(* Logix 5000 project; controller PRU vendor 1 type 14 code 107 rev 20.13; software revision 20.01; part 16 of 17 *)
(* tags used below, declared in another part *)
   ABS_ENCODER_ERROR_MINUS : REAL;
   ABS_ENCODER_ERROR_PLUS : REAL;
   ACCEL_DECEL_RAMP : REAL;   // VFD Accel/Decel ramp rate * 10ms ie 100 * 10ms = 1sec
   ACTUAL_FWD_ION : BOOL;
   ACTUAL_ILLEGAL_ION : BOOL;
   ACTUAL_REV_ION : BOOL;
   AFI : BOOL;
   AUTO_FWD_CMD : BOOL;
   AUTO_FWD_CMD_GON : BOOL;
   AUTO_FWD_CMD_GON_VALUE : DINT;
   AUTO_FWD_CMD_VALUE : DINT;
   CENTERING_BON : BOOL;
   CENTERING_BON_ONS : BOOL;
   CENTERING_BON_SS : BOOL;
   CENTERING_ERROR : REAL;
   CENTERING_ERROR_NOW : REAL;
   CENTERING_ERROR_WAS : REAL;
   CENTERING_ONS : BOOL;
   CENTERING_SS : BOOL;
   CENTERING_TON : TIMER;
   CR7_VFD_DRYERL_GON : BOOL;
   CR7_VFD_DRYERL_LON : BOOL;
   DATA_RECORD_INDEX : INT;
   DRYER : DUAL_SCREW;
   DRYER_CENTER_STARTUP_MODE : BOOL;
   DRYER_IS_CENTERING : BOOL;
   DRYER_MODE_AUTO : BOOL;
   DRYERL_ACTUAL_SPEED : REAL;
   DRYERR_ACTUAL_SPEED : REAL;
   ENCODER_ACC : REAL;
   ENCODER_ERROR : REAL;
   ENCODER_OFFSET : REAL;
   ENCODER_RATE : REAL;
   ESR_CONTACT_1_ION : BOOL;
   ESR_CONTACT_2_ION : BOOL;
   ESR_RESET_PB_ION : BOOL;
   FAULT : DINT[100];
   FAULT_31_14_ONS : BOOL;
   FAULT_TIMER : TIMER[10000];
   FAULT_TIMER_3112_TmrExtended : BOOL;
   FAULT_TIMER_3112_TmrNormal : BOOL;
   FAULTS_FA1_IOK : BOOL;   // SYSTEM LEVEL FAULTS ARE OK.
   FAULTS_FA1B_IOK : BOOL;   // STOP PUSHBUTTON FAULTS ARE OK.
   FAULTS_FA3_IOK : BOOL;
   FAULTS_FA3A_IOK : BOOL;   // SCREWS DRIVES NOT FAULTED.
   FAULTS_FA3B_IOK : BOOL;   // ENCODERS NOT FAULTED.
   FEED_TIME_OFF : TIMER;
   FEED_TIME_OFF_REM : REAL;
   FEED_TIME_OFF_REM_TEMP : REAL;
   FEED_TIME_OFF_SEC : REAL;
   FEED_TIME_ON : TIMER;
   FEED_TIME_ON_REM : REAL;
   FEED_TIME_ON_REM_TEMP : REAL;
   FEED_TIME_ON_SEC : REAL;
   FEED_TRIGGER : BOOL;
   FWD_CMD_BON : TIMER;
   GRAY : REAL[4097];
   HMI_ALARM_RESET : BOOL;
   HMI_AUTO_SETPOINT_FDBK : REAL;
   HMI_CR7_FORCE_OFF : BOOL;
   HMI_CR7_FORCE_ON : BOOL;
   HMI_DCS_SPEED_FDBK : REAL;
   HMI_DSC_SPEED_CMD : REAL;
   HMI_FINAL_SCREW_POSITION_ERROR : REAL;
   HMI_OSC_INC : REAL;
   HMI_WIPER_OSC_SETPOINT : REAL;
   HMI_ZERO_SPEED_FORCE_ION : BOOL;
   INTERRUPT_INDEX : INT;
   LEFT_AUTO_PCNT_SETPOINT : REAL;
   LEFT_RATE : REAL;
   MASTER_RIGHT_CMD : BOOL;
   MAX_ENCODER_ERROR_MINUS : REAL;
   MAX_ENCODER_ERROR_PLUS : REAL;
   MIX_FWD_PRESET : REAL;
   MIX_MODE_TIMEBASE : BOOL;
   MIX_REV_PER_MIN : REAL;
   MIX_REV_PRESET : REAL;
   MODE_DRYER : INT;
   OK_TO_CHANGE_DIR : BOOL;
   OK_TO_STOP : BOOL;
   PF70EL_Message : MESSAGE;
   PF70ER_Message : MESSAGE;
   RAMP_COUNT : DINT;
   RAMP_TIME : DINT;
   RAMPING_SPEED_DOWN : BOOL;
   RAMPING_SPEED_UP : BOOL;
   RelaxEncoderFaultTime_SpeedSP : REAL;
   RelaxEncoderFaultTime_SpeedSP_Rev : REAL;
   RETENTION_TIME_MIN : REAL;
   REV_CMD_BON : TIMER;
   RIGHT_AUTO_PCNT_SETPOINT : REAL;
   RIGHT_RATE : REAL;
   SCREW_ENCODERS : SCREW_ENCODERS;
   SCREW_PITCH_CONSTANT : REAL;
   SCREW_SPEED : SCREW_SPEED;
   SCREW_SPEED_OUT_L : REAL;
   SCREW_SPEED_OUT_R : REAL;
   SCREW_WIPE : SCREW_WIPER;
   SCREWS_ENABLE_GON : BOOL;   // Dryer screw faults are ok.
   SCREWS_WIPE_HOLD_TIME : DINT;
   SET_PYRO_SPEED_TO_ZERO : BOOL;
   SLAVE_COMP_LIMIT : REAL;
   SPEED_RAMP_FREEZE_TOF : TIMER;
   SPEED_RAMP_MULT : REAL;
   VFD_1_Current : DINT;
   VFD_1_Current_Real : REAL;
   VFD_1_Tot : EnergyTot;   // Left Dryer
   VFD_2_Current : DINT;
   VFD_2_Current_Real : REAL;
   VFD_2_Tot : EnergyTot;   // Right Dryer
   VFDS_BON : BOOL;   // DRYER VFDs HAVE BEEN COMMANDED ON FOR 1 SECOND.
   WIPE_ACTUAL : REAL;
   WIPE_EON : BOOL;
   WIPE_FREEZE_CMD : BOOL;
   WIPE_HOLDING : BOOL;
   WIPE_MASTER : BOOL;
   WIPE_MASTER_BOF : TIMER;
   WIPE_MASTER_BON : TIMER;
   WIPE_MASTER_ONS : BOOL;
   WIPE_MASTER_SS : BOOL;
   WIPE_PERIOD_COUNTS_ACC : REAL;
   WIPE_PERIOD_ONS : BOOL;
   WIPE_PERIOD_SECONDS : REAL;
   WIPE_TON : TIMER;
(* SCREW_CONTROL, continued *)

ROUTINE B03_FA3_B_ENCODER_FAULTS_3100   (* ladder *)
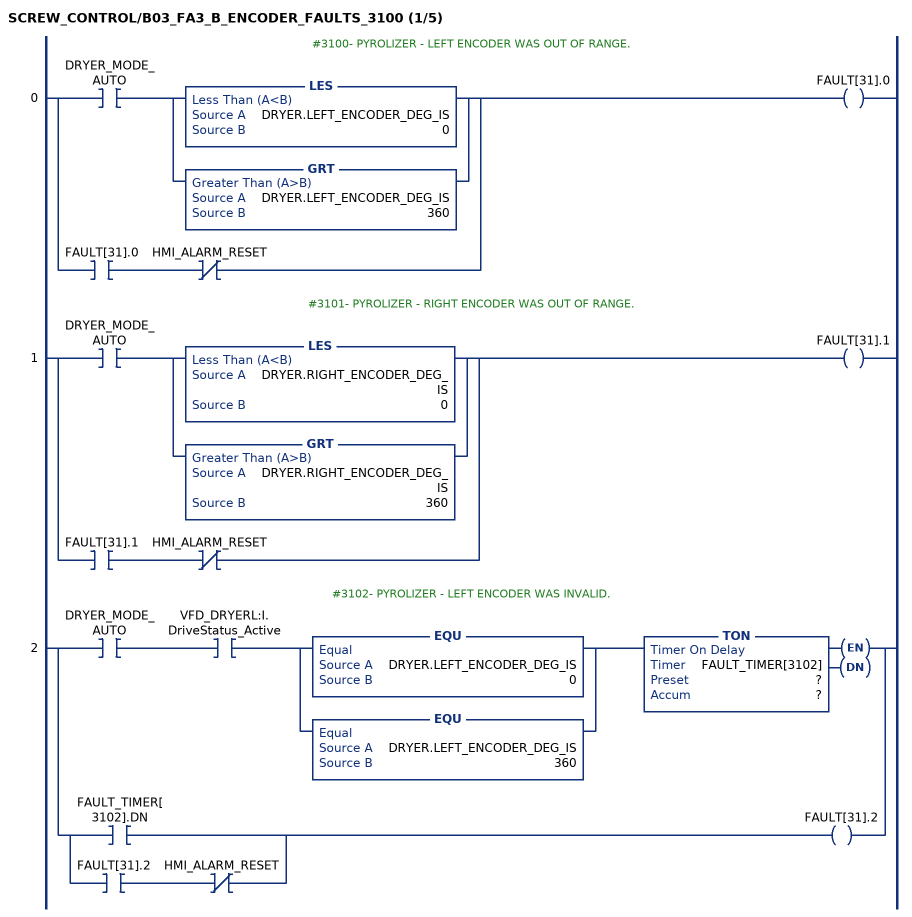
   // #3100- PYROLIZER - LEFT ENCODER WAS OUT OF RANGE.
   0: [XIC(DRYER_MODE_AUTO) [LES(DRYER.LEFT_ENCODER_DEG_IS,0) ,GRT(DRYER.LEFT_ENCODER_DEG_IS,360) ] ,XIC(FAULT[31].0) XIO(HMI_ALARM_RESET) ]OTE(FAULT[31].0);
   // #3101- PYROLIZER - RIGHT ENCODER WAS OUT OF RANGE.
   1: [XIC(DRYER_MODE_AUTO) [LES(DRYER.RIGHT_ENCODER_DEG_IS,0) ,GRT(DRYER.RIGHT_ENCODER_DEG_IS,360) ] ,XIC(FAULT[31].1) XIO(HMI_ALARM_RESET) ]OTE(FAULT[31].1);
   // #3102- PYROLIZER - LEFT ENCODER WAS INVALID.
   2: [XIC(DRYER_MODE_AUTO) XIC(VFD_DRYERL:I.DriveStatus_Active) [EQU(DRYER.LEFT_ENCODER_DEG_IS,0) ,EQU(DRYER.LEFT_ENCODER_DEG_IS,360) ] TON(FAULT_TIMER[3102],?,?) ,[XIC(FAULT_TIMER[3102].DN) ,XIC(FAULT[31].2) XIO(HMI_ALARM_RESET) ] OTE(FAULT[31].2) ];
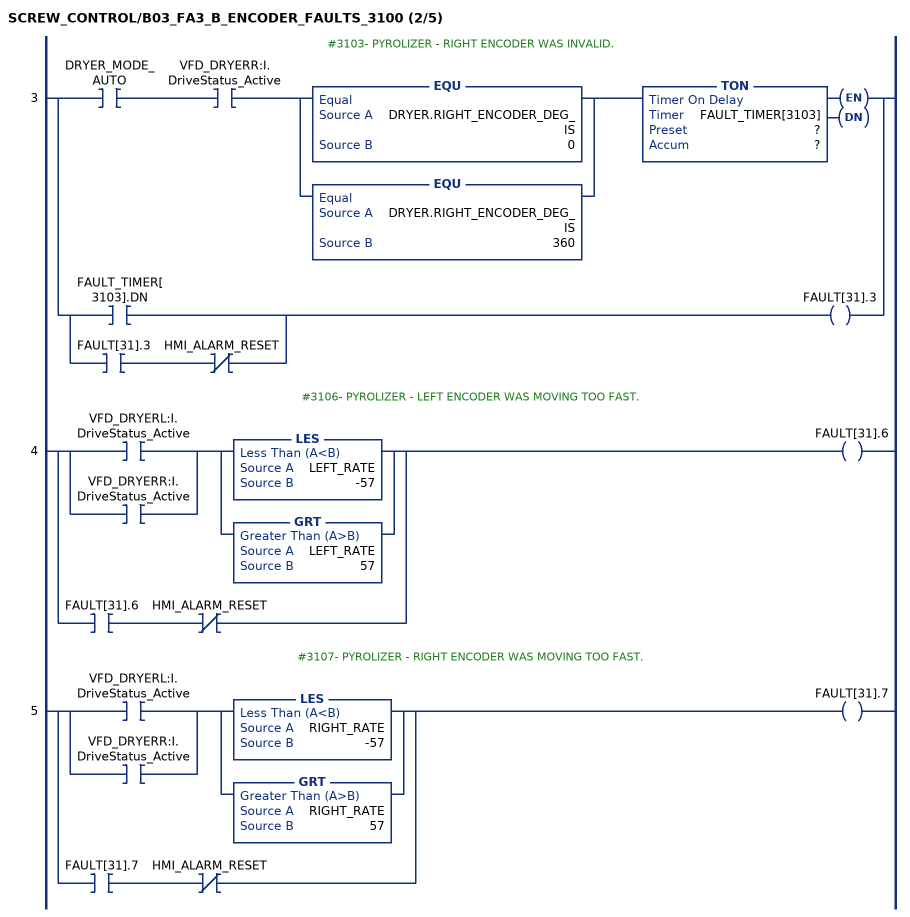
   // #3103- PYROLIZER - RIGHT ENCODER WAS INVALID.
   3: [XIC(DRYER_MODE_AUTO) XIC(VFD_DRYERR:I.DriveStatus_Active) [EQU(DRYER.RIGHT_ENCODER_DEG_IS,0) ,EQU(DRYER.RIGHT_ENCODER_DEG_IS,360) ] TON(FAULT_TIMER[3103],?,?) ,[XIC(FAULT_TIMER[3103].DN) ,XIC(FAULT[31].3) XIO(HMI_ALARM_RESET) ] OTE(FAULT[31].3) ];
   // #3106- PYROLIZER - LEFT ENCODER WAS MOVING TOO FAST.
   4: [[XIC(VFD_DRYERL:I.DriveStatus_Active) ,XIC(VFD_DRYERR:I.DriveStatus_Active) ] [LES(LEFT_RATE,-57) ,GRT(LEFT_RATE,57) ] ,XIC(FAULT[31].6) XIO(HMI_ALARM_RESET) ]OTE(FAULT[31].6);
   // #3107- PYROLIZER - RIGHT ENCODER WAS MOVING TOO FAST.
   5: [[XIC(VFD_DRYERL:I.DriveStatus_Active) ,XIC(VFD_DRYERR:I.DriveStatus_Active) ] [LES(RIGHT_RATE,-57) ,GRT(RIGHT_RATE,57) ] ,XIC(FAULT[31].7) XIO(HMI_ALARM_RESET) ]OTE(FAULT[31].7);
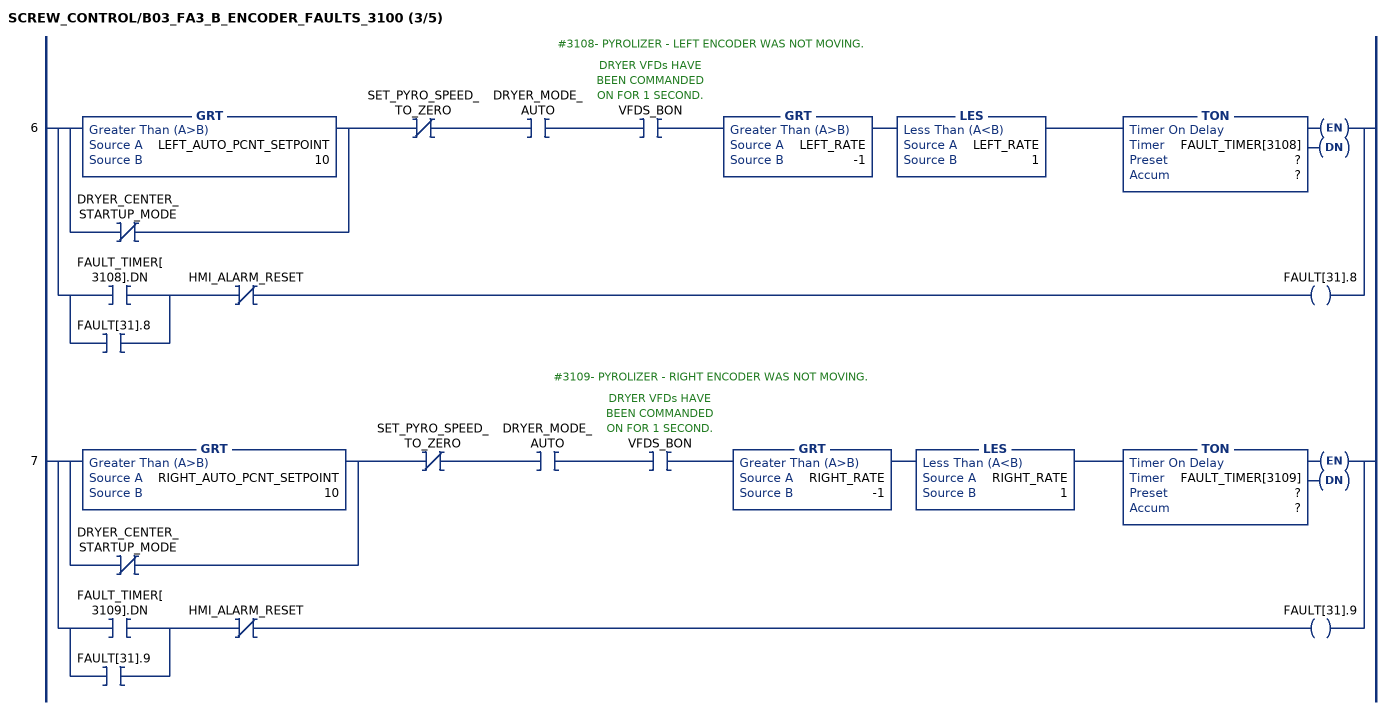
   // #3108- PYROLIZER - LEFT ENCODER WAS NOT MOVING.
   6: [[GRT(LEFT_AUTO_PCNT_SETPOINT,10) ,XIO(DRYER_CENTER_STARTUP_MODE) ] XIO(SET_PYRO_SPEED_TO_ZERO) XIC(DRYER_MODE_AUTO) XIC(VFDS_BON) GRT(LEFT_RATE,-1) LES(LEFT_RATE,1) TON(FAULT_TIMER[3108],?,?) ,[XIC(FAULT_TIMER[3108].DN) ,XIC(FAULT[31].8) ] XIO(HMI_ALARM_RESET) OTE(FAULT[31].8) ];
   // #3109- PYROLIZER - RIGHT ENCODER WAS NOT MOVING.
   7: [[GRT(RIGHT_AUTO_PCNT_SETPOINT,10) ,XIO(DRYER_CENTER_STARTUP_MODE) ] XIO(SET_PYRO_SPEED_TO_ZERO) XIC(DRYER_MODE_AUTO) XIC(VFDS_BON) GRT(RIGHT_RATE,-1) LES(RIGHT_RATE,1) TON(FAULT_TIMER[3109],?,?) ,[XIC(FAULT_TIMER[3109].DN) ,XIC(FAULT[31].9) ] XIO(HMI_ALARM_RESET) OTE(FAULT[31].9) ];
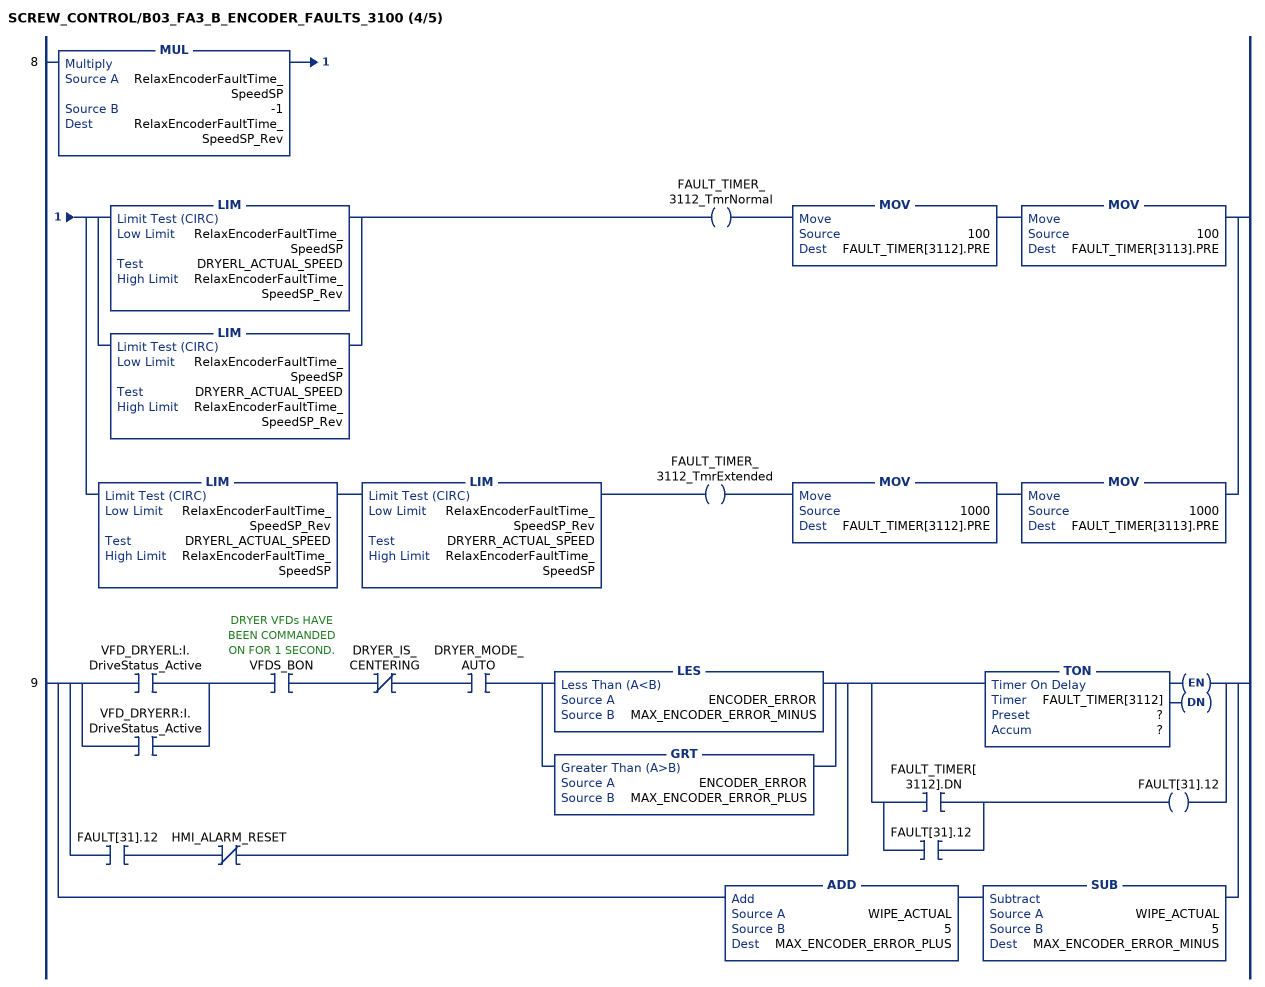
   8: MUL(RelaxEncoderFaultTime_SpeedSP,-1,RelaxEncoderFaultTime_SpeedSP_Rev)[[LIM(RelaxEncoderFaultTime_SpeedSP,DRYERL_ACTUAL_SPEED,RelaxEncoderFaultTime_SpeedSP_Rev) ,LIM(RelaxEncoderFaultTime_SpeedSP,DRYERR_ACTUAL_SPEED,RelaxEncoderFaultTime_SpeedSP_Rev) ] OTE(FAULT_TIMER_3112_TmrNormal) MOV(100,FAULT_TIMER[3112].PRE) MOV(100,FAULT_TIMER[3113].PRE) ,LIM(RelaxEncoderFaultTime_SpeedSP_Rev,DRYERL_ACTUAL_SPEED,RelaxEncoderFaultTime_SpeedSP) LIM(RelaxEncoderFaultTime_SpeedSP_Rev,DRYERR_ACTUAL_SPEED,RelaxEncoderFaultTime_SpeedSP) OTE(FAULT_TIMER_3112_TmrExtended) MOV(1000,FAULT_TIMER[3112].PRE) MOV(1000,FAULT_TIMER[3113].PRE) ];
   9: [[[XIC(VFD_DRYERL:I.DriveStatus_Active) ,XIC(VFD_DRYERR:I.DriveStatus_Active) ] XIC(VFDS_BON) XIO(DRYER_IS_CENTERING) XIC(DRYER_MODE_AUTO) [LES(ENCODER_ERROR,MAX_ENCODER_ERROR_MINUS) ,GRT(ENCODER_ERROR,MAX_ENCODER_ERROR_PLUS) ] ,XIC(FAULT[31].12) XIO(HMI_ALARM_RESET) ] [TON(FAULT_TIMER[3112],?,?) ,[XIC(FAULT_TIMER[3112].DN) ,XIC(FAULT[31].12) ] OTE(FAULT[31].12) ] ,ADD(WIPE_ACTUAL,5,MAX_ENCODER_ERROR_PLUS) SUB(WIPE_ACTUAL,5,MAX_ENCODER_ERROR_MINUS) ];
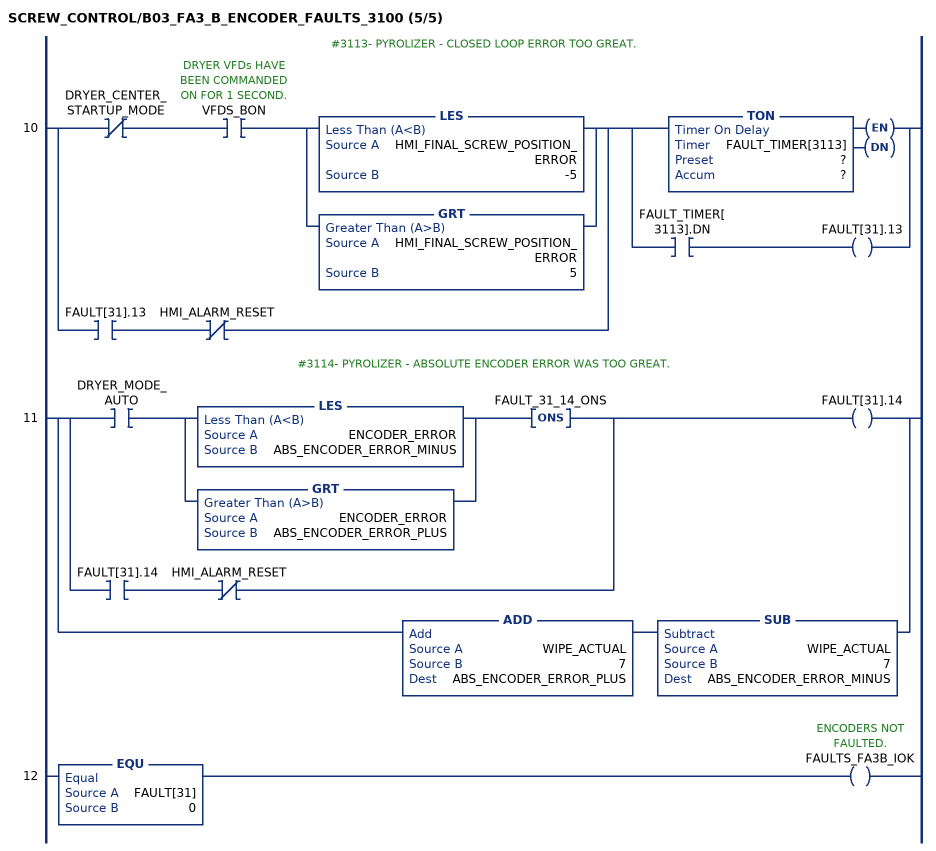
   // #3113- PYROLIZER - CLOSED LOOP ERROR TOO GREAT.
   10: [XIO(DRYER_CENTER_STARTUP_MODE) XIC(VFDS_BON) [LES(HMI_FINAL_SCREW_POSITION_ERROR,-5) ,GRT(HMI_FINAL_SCREW_POSITION_ERROR,5) ] ,XIC(FAULT[31].13) XIO(HMI_ALARM_RESET) ][TON(FAULT_TIMER[3113],?,?) ,XIC(FAULT_TIMER[3113].DN) OTE(FAULT[31].13) ];
   // #3114- PYROLIZER - ABSOLUTE ENCODER ERROR WAS TOO GREAT.
   11: [[XIC(DRYER_MODE_AUTO) [LES(ENCODER_ERROR,ABS_ENCODER_ERROR_MINUS) ,GRT(ENCODER_ERROR,ABS_ENCODER_ERROR_PLUS) ] ONS(FAULT_31_14_ONS) ,XIC(FAULT[31].14) XIO(HMI_ALARM_RESET) ] OTE(FAULT[31].14) ,ADD(WIPE_ACTUAL,7,ABS_ENCODER_ERROR_PLUS) SUB(WIPE_ACTUAL,7,ABS_ENCODER_ERROR_MINUS) ];
   12: EQU(FAULT[31],0)OTE(FAULTS_FA3B_IOK);
END_ROUTINE

ROUTINE DUALSCREW   (* ladder *)
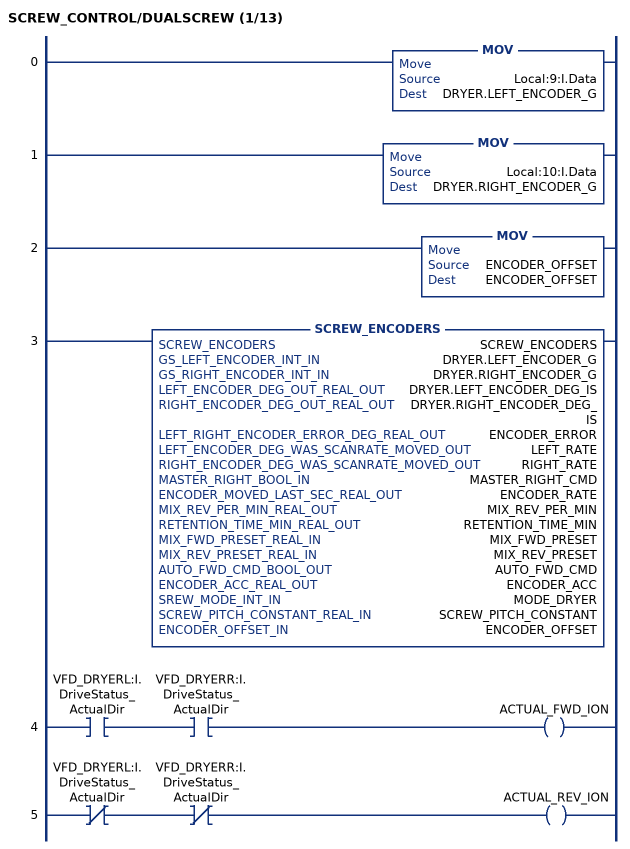
   0: MOV(Local:9:I.Data,DRYER.LEFT_ENCODER_G);
   1: MOV(Local:10:I.Data,DRYER.RIGHT_ENCODER_G);
   2: MOV(ENCODER_OFFSET,ENCODER_OFFSET);
   3: SCREW_ENCODERS(SCREW_ENCODERS,DRYER.LEFT_ENCODER_G,DRYER.RIGHT_ENCODER_G,DRYER.LEFT_ENCODER_DEG_IS,DRYER.RIGHT_ENCODER_DEG_IS,ENCODER_ERROR,LEFT_RATE,RIGHT_RATE,MASTER_RIGHT_CMD,ENCODER_RATE,MIX_REV_PER_MIN,RETENTION_TIME_MIN,MIX_FWD_PRESET,MIX_REV_PRESET,AUTO_FWD_CMD,ENCODER_ACC,MODE_DRYER,SCREW_PITCH_CONSTANT,ENCODER_OFFSET);
   4: XIC(VFD_DRYERL:I.DriveStatus_ActualDir)XIC(VFD_DRYERR:I.DriveStatus_ActualDir)OTE(ACTUAL_FWD_ION);
   5: XIO(VFD_DRYERL:I.DriveStatus_ActualDir)XIO(VFD_DRYERR:I.DriveStatus_ActualDir)OTE(ACTUAL_REV_ION);
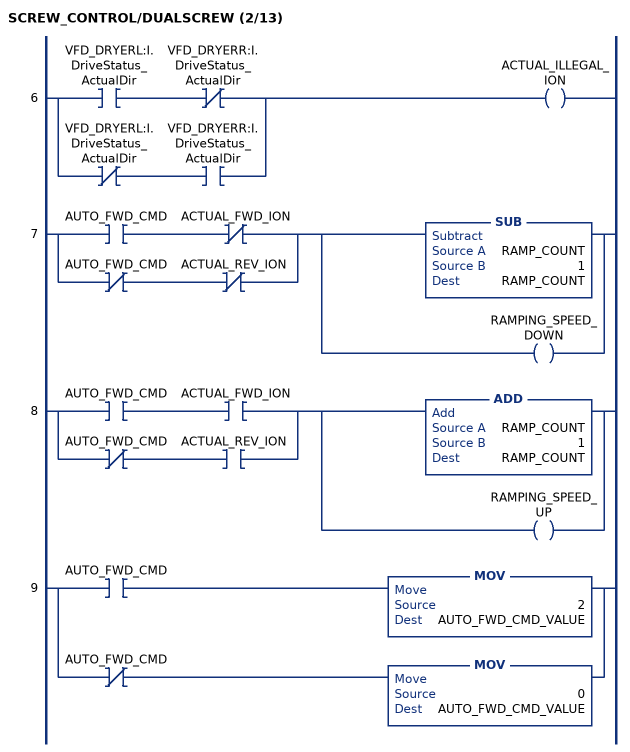
   6: [XIC(VFD_DRYERL:I.DriveStatus_ActualDir) XIO(VFD_DRYERR:I.DriveStatus_ActualDir) ,XIO(VFD_DRYERL:I.DriveStatus_ActualDir) XIC(VFD_DRYERR:I.DriveStatus_ActualDir) ]OTE(ACTUAL_ILLEGAL_ION);
   7: [XIC(AUTO_FWD_CMD) XIO(ACTUAL_FWD_ION) ,XIO(AUTO_FWD_CMD) XIO(ACTUAL_REV_ION) ][SUB(RAMP_COUNT,1,RAMP_COUNT) ,OTE(RAMPING_SPEED_DOWN) ];
   8: [XIC(AUTO_FWD_CMD) XIC(ACTUAL_FWD_ION) ,XIO(AUTO_FWD_CMD) XIC(ACTUAL_REV_ION) ][ADD(RAMP_COUNT,1,RAMP_COUNT) ,OTE(RAMPING_SPEED_UP) ];
   9: [XIC(AUTO_FWD_CMD) MOV(2,AUTO_FWD_CMD_VALUE) ,XIO(AUTO_FWD_CMD) MOV(0,AUTO_FWD_CMD_VALUE) ];
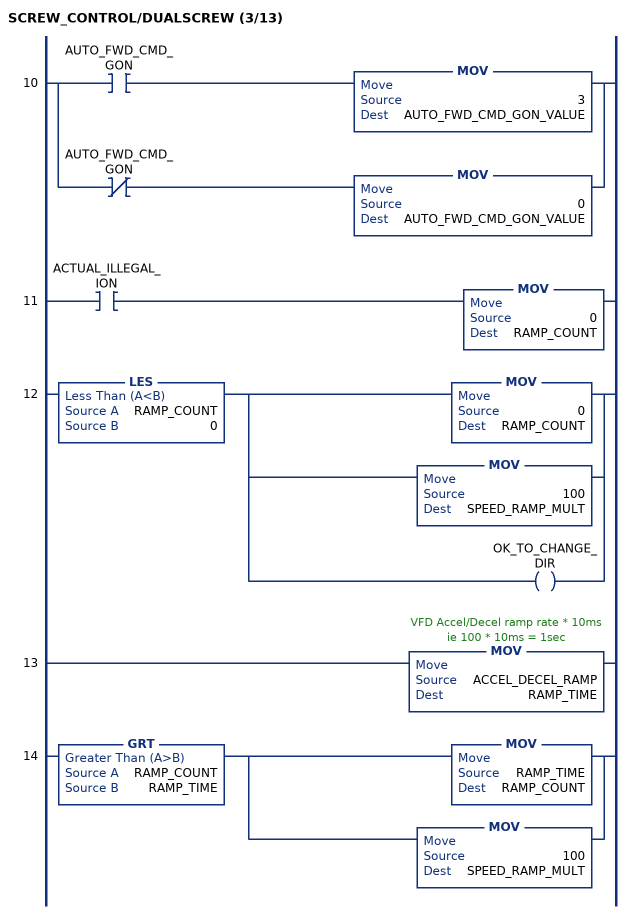
   10: [XIC(AUTO_FWD_CMD_GON) MOV(3,AUTO_FWD_CMD_GON_VALUE) ,XIO(AUTO_FWD_CMD_GON) MOV(0,AUTO_FWD_CMD_GON_VALUE) ];
   11: XIC(ACTUAL_ILLEGAL_ION)MOV(0,RAMP_COUNT);
   12: LES(RAMP_COUNT,0)[MOV(0,RAMP_COUNT) ,MOV(100,SPEED_RAMP_MULT) ,OTE(OK_TO_CHANGE_DIR) ];
   13: MOV(ACCEL_DECEL_RAMP,RAMP_TIME);
   14: GRT(RAMP_COUNT,RAMP_TIME)[MOV(RAMP_TIME,RAMP_COUNT) ,MOV(100,SPEED_RAMP_MULT) ];
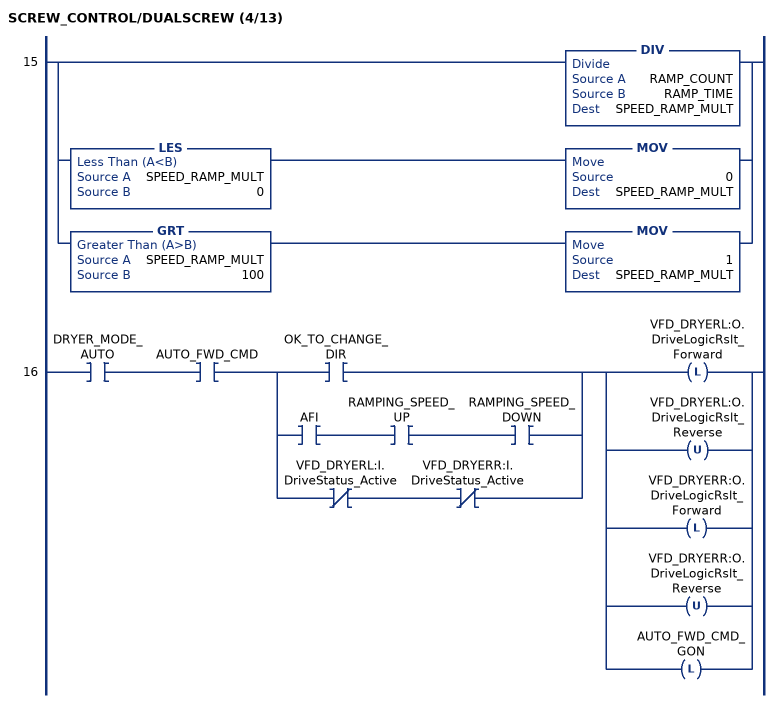
   15: [DIV(RAMP_COUNT,RAMP_TIME,SPEED_RAMP_MULT) ,LES(SPEED_RAMP_MULT,0) MOV(0,SPEED_RAMP_MULT) ,GRT(SPEED_RAMP_MULT,100) MOV(1,SPEED_RAMP_MULT) ];
   16: XIC(DRYER_MODE_AUTO)XIC(AUTO_FWD_CMD)[XIC(OK_TO_CHANGE_DIR) ,XIC(AFI) XIC(RAMPING_SPEED_UP) XIC(RAMPING_SPEED_DOWN) ,XIO(VFD_DRYERL:I.DriveStatus_Active) XIO(VFD_DRYERR:I.DriveStatus_Active) ][OTL(VFD_DRYERL:O.DriveLogicRslt_Forward) ,OTU(VFD_DRYERL:O.DriveLogicRslt_Reverse) ,OTL(VFD_DRYERR:O.DriveLogicRslt_Forward) ,OTU(VFD_DRYERR:O.DriveLogicRslt_Reverse) ,OTL(AUTO_FWD_CMD_GON) ];
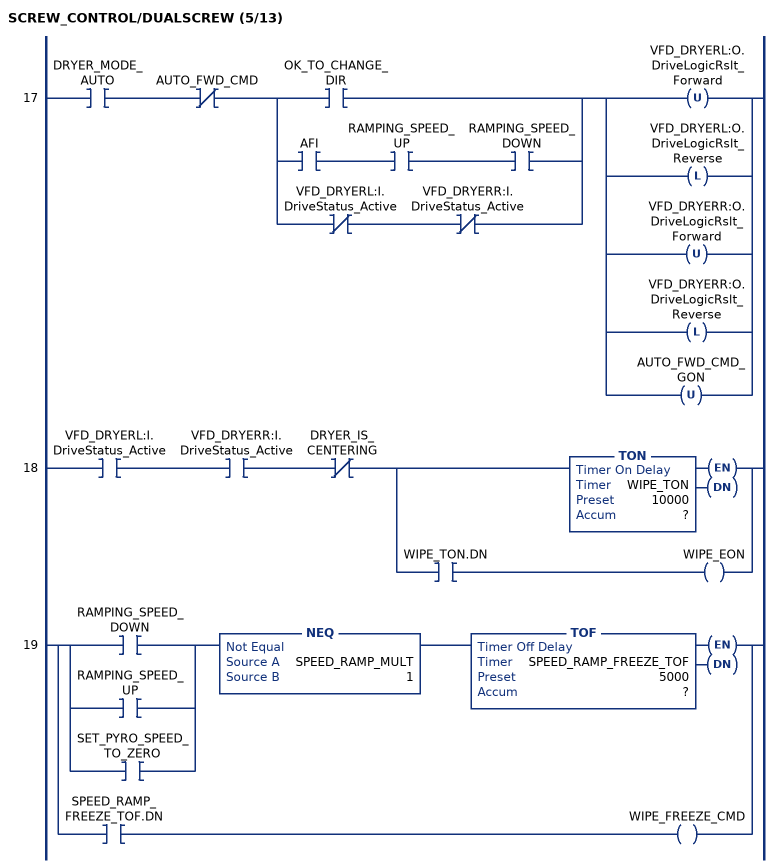
   17: XIC(DRYER_MODE_AUTO)XIO(AUTO_FWD_CMD)[XIC(OK_TO_CHANGE_DIR) ,XIC(AFI) XIC(RAMPING_SPEED_UP) XIC(RAMPING_SPEED_DOWN) ,XIO(VFD_DRYERL:I.DriveStatus_Active) XIO(VFD_DRYERR:I.DriveStatus_Active) ][OTU(VFD_DRYERL:O.DriveLogicRslt_Forward) ,OTL(VFD_DRYERL:O.DriveLogicRslt_Reverse) ,OTU(VFD_DRYERR:O.DriveLogicRslt_Forward) ,OTL(VFD_DRYERR:O.DriveLogicRslt_Reverse) ,OTU(AUTO_FWD_CMD_GON) ];
   18: XIC(VFD_DRYERL:I.DriveStatus_Active)XIC(VFD_DRYERR:I.DriveStatus_Active)XIO(DRYER_IS_CENTERING)[TON(WIPE_TON,?,?) ,XIC(WIPE_TON.DN) OTE(WIPE_EON) ];
   19: [[XIC(RAMPING_SPEED_DOWN) ,XIC(RAMPING_SPEED_UP) ,XIC(SET_PYRO_SPEED_TO_ZERO) ] NEQ(SPEED_RAMP_MULT,1) TOF(SPEED_RAMP_FREEZE_TOF,?,?) ,XIC(SPEED_RAMP_FREEZE_TOF.DN) OTE(WIPE_FREEZE_CMD) ];
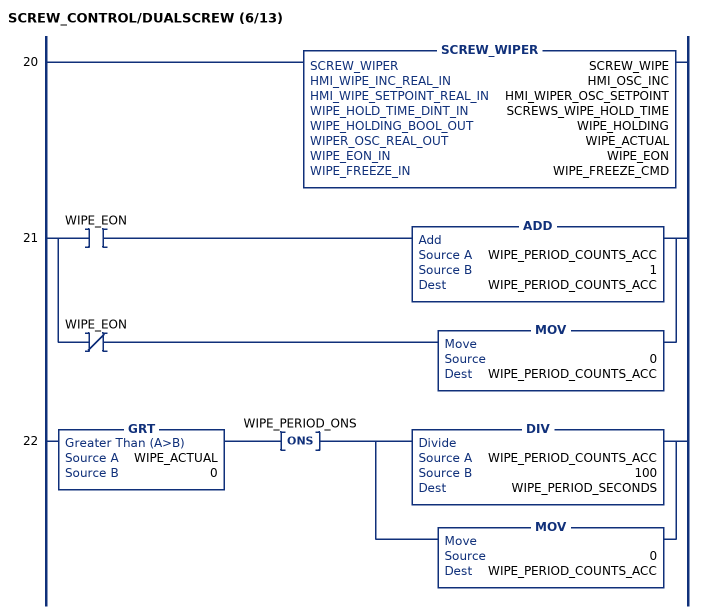
   20: SCREW_WIPER(SCREW_WIPE,HMI_OSC_INC,HMI_WIPER_OSC_SETPOINT,SCREWS_WIPE_HOLD_TIME,WIPE_HOLDING,WIPE_ACTUAL,WIPE_EON,WIPE_FREEZE_CMD);
   21: [XIC(WIPE_EON) ADD(WIPE_PERIOD_COUNTS_ACC,1,WIPE_PERIOD_COUNTS_ACC) ,XIO(WIPE_EON) MOV(0,WIPE_PERIOD_COUNTS_ACC) ];
   22: GRT(WIPE_ACTUAL,0)ONS(WIPE_PERIOD_ONS)[DIV(WIPE_PERIOD_COUNTS_ACC,100,WIPE_PERIOD_SECONDS) ,MOV(0,WIPE_PERIOD_COUNTS_ACC) ];
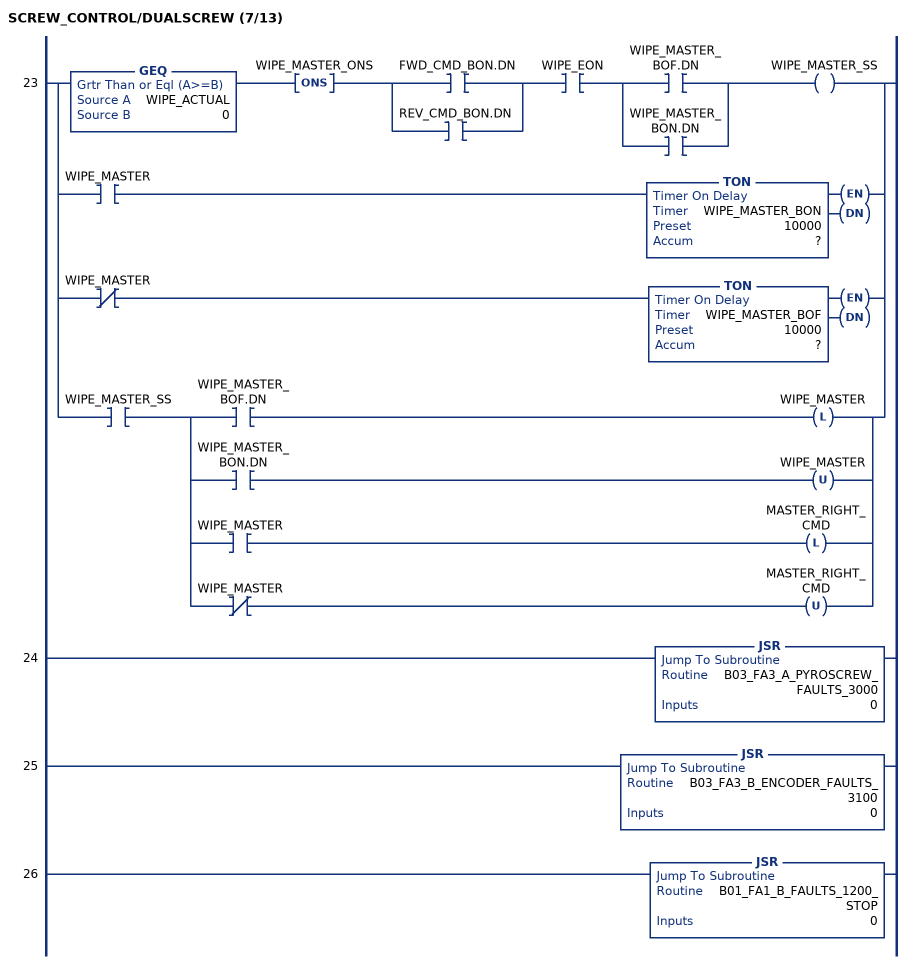
   23: [GEQ(WIPE_ACTUAL,0) ONS(WIPE_MASTER_ONS) [XIC(FWD_CMD_BON.DN) ,XIC(REV_CMD_BON.DN) ] XIC(WIPE_EON) [XIC(WIPE_MASTER_BOF.DN) ,XIC(WIPE_MASTER_BON.DN) ] OTE(WIPE_MASTER_SS) ,XIC(WIPE_MASTER) TON(WIPE_MASTER_BON,?,?) ,XIO(WIPE_MASTER) TON(WIPE_MASTER_BOF,?,?) ,XIC(WIPE_MASTER_SS) [XIC(WIPE_MASTER_BOF.DN) OTL(WIPE_MASTER) ,XIC(WIPE_MASTER_BON.DN) OTU(WIPE_MASTER) ,XIC(WIPE_MASTER) OTL(MASTER_RIGHT_CMD) ,XIO(WIPE_MASTER) OTU(MASTER_RIGHT_CMD) ] ];
   24: JSR(B03_FA3_A_PYROSCREW_FAULTS_3000,0);
   25: JSR(B03_FA3_B_ENCODER_FAULTS_3100,0);
   26: JSR(B01_FA1_B_FAULTS_1200_STOP,0);
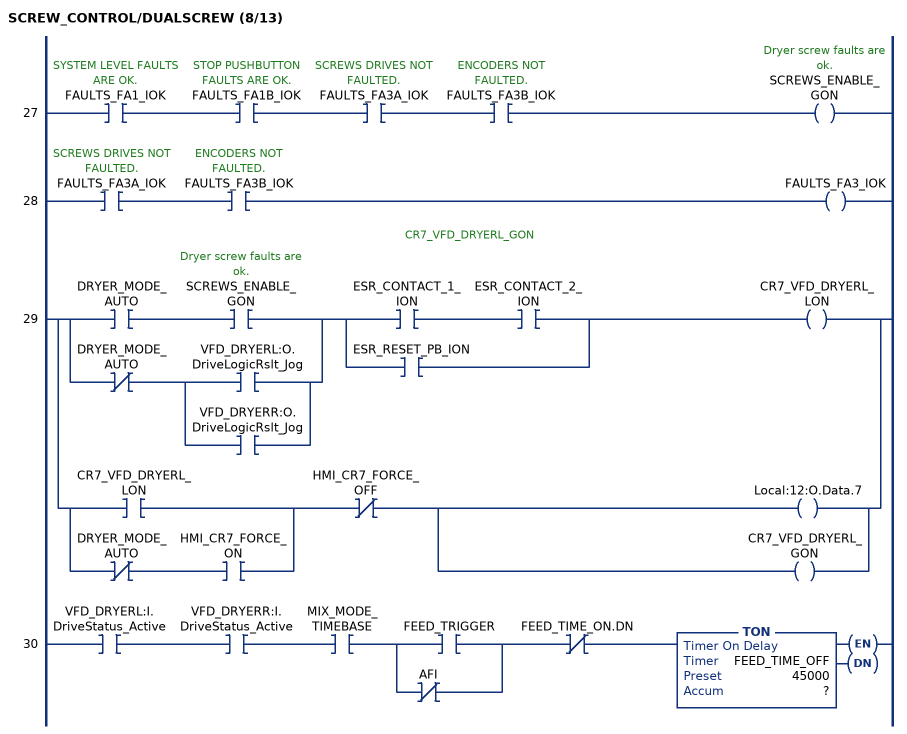
   27: XIC(FAULTS_FA1_IOK)XIC(FAULTS_FA1B_IOK)XIC(FAULTS_FA3A_IOK)XIC(FAULTS_FA3B_IOK)OTE(SCREWS_ENABLE_GON);
   28: XIC(FAULTS_FA3A_IOK)XIC(FAULTS_FA3B_IOK)OTE(FAULTS_FA3_IOK);
   // CR7_VFD_DRYERL_GON
   29: [[XIC(DRYER_MODE_AUTO) XIC(SCREWS_ENABLE_GON) ,XIO(DRYER_MODE_AUTO) [XIC(VFD_DRYERL:O.DriveLogicRslt_Jog) ,XIC(VFD_DRYERR:O.DriveLogicRslt_Jog) ] ] [XIC(ESR_CONTACT_1_ION) XIC(ESR_CONTACT_2_ION) ,XIC(ESR_RESET_PB_ION) ] OTE(CR7_VFD_DRYERL_LON) ,[XIC(CR7_VFD_DRYERL_LON) ,XIO(DRYER_MODE_AUTO) XIC(HMI_CR7_FORCE_ON) ] XIO(HMI_CR7_FORCE_OFF) [OTE(Local:12:O.Data.7) ,OTE(CR7_VFD_DRYERL_GON) ] ];
   30: XIC(VFD_DRYERL:I.DriveStatus_Active)XIC(VFD_DRYERR:I.DriveStatus_Active)XIC(MIX_MODE_TIMEBASE)[XIC(FEED_TRIGGER) ,XIO(AFI) ]XIO(FEED_TIME_ON.DN)TON(FEED_TIME_OFF,?,?);
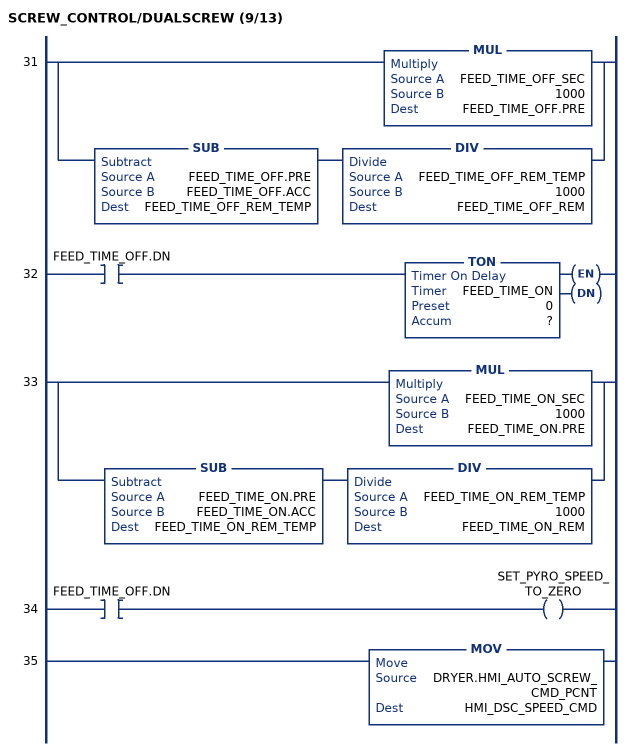
   31: [MUL(FEED_TIME_OFF_SEC,1000,FEED_TIME_OFF.PRE) ,SUB(FEED_TIME_OFF.PRE,FEED_TIME_OFF.ACC,FEED_TIME_OFF_REM_TEMP) DIV(FEED_TIME_OFF_REM_TEMP,1000,FEED_TIME_OFF_REM) ];
   32: XIC(FEED_TIME_OFF.DN)TON(FEED_TIME_ON,?,?);
   33: [MUL(FEED_TIME_ON_SEC,1000,FEED_TIME_ON.PRE) ,SUB(FEED_TIME_ON.PRE,FEED_TIME_ON.ACC,FEED_TIME_ON_REM_TEMP) DIV(FEED_TIME_ON_REM_TEMP,1000,FEED_TIME_ON_REM) ];
   34: XIC(FEED_TIME_OFF.DN)OTE(SET_PYRO_SPEED_TO_ZERO);
   35: MOV(DRYER.HMI_AUTO_SCREW_CMD_PCNT,HMI_DSC_SPEED_CMD);
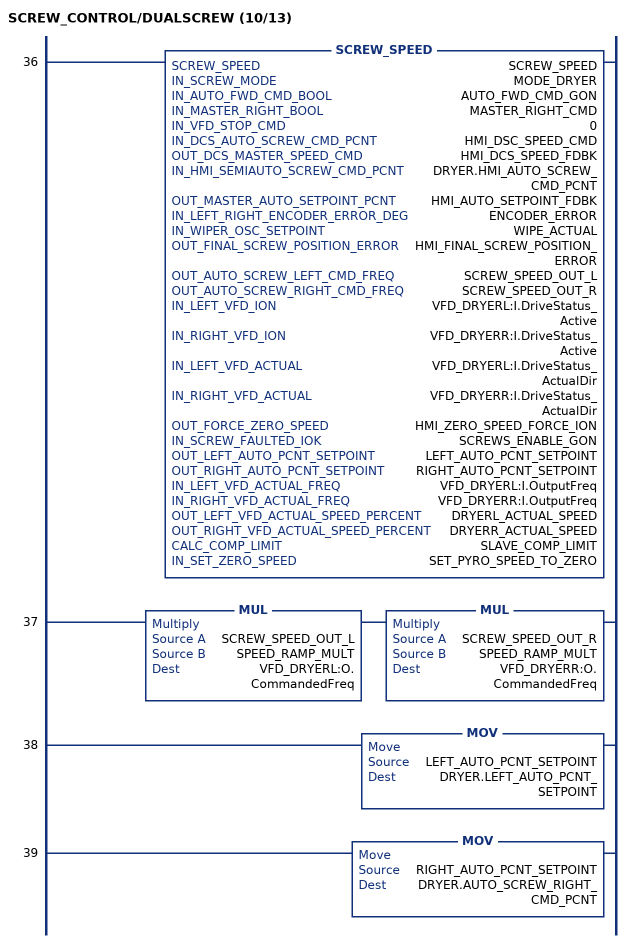
   36: SCREW_SPEED(SCREW_SPEED,MODE_DRYER,AUTO_FWD_CMD_GON,MASTER_RIGHT_CMD,0,HMI_DSC_SPEED_CMD,HMI_DCS_SPEED_FDBK,DRYER.HMI_AUTO_SCREW_CMD_PCNT,HMI_AUTO_SETPOINT_FDBK,ENCODER_ERROR,WIPE_ACTUAL,HMI_FINAL_SCREW_POSITION_ERROR,SCREW_SPEED_OUT_L,SCREW_SPEED_OUT_R,VFD_DRYERL:I.DriveStatus_Active,VFD_DRYERR:I.DriveStatus_Active,VFD_DRYERL:I.DriveStatus_ActualDir,VFD_DRYERR:I.DriveStatus_ActualDir,HMI_ZERO_SPEED_FORCE_ION,SCREWS_ENABLE_GON,LEFT_AUTO_PCNT_SETPOINT,RIGHT_AUTO_PCNT_SETPOINT,VFD_DRYERL:I.OutputFreq,VFD_DRYERR:I.OutputFreq,DRYERL_ACTUAL_SPEED,DRYERR_ACTUAL_SPEED,SLAVE_COMP_LIMIT,SET_PYRO_SPEED_TO_ZERO);
   37: MUL(SCREW_SPEED_OUT_L,SPEED_RAMP_MULT,VFD_DRYERL:O.CommandedFreq)MUL(SCREW_SPEED_OUT_R,SPEED_RAMP_MULT,VFD_DRYERR:O.CommandedFreq);
   38: MOV(LEFT_AUTO_PCNT_SETPOINT,DRYER.LEFT_AUTO_PCNT_SETPOINT);
   39: MOV(RIGHT_AUTO_PCNT_SETPOINT,DRYER.AUTO_SCREW_RIGHT_CMD_PCNT);
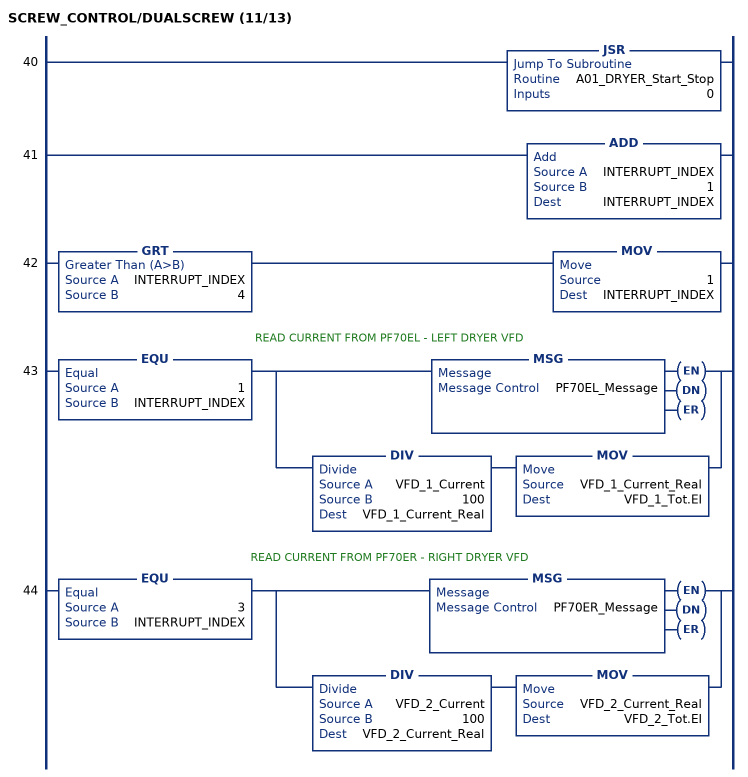
   40: JSR(A01_DRYER_Start_Stop,0);
   41: ADD(INTERRUPT_INDEX,1,INTERRUPT_INDEX);
   42: GRT(INTERRUPT_INDEX,4)MOV(1,INTERRUPT_INDEX);
   // READ CURRENT FROM PF70EL - LEFT DRYER VFD
   43: EQU(1,INTERRUPT_INDEX)[MSG(PF70EL_Message) ,DIV(VFD_1_Current,100,VFD_1_Current_Real) MOV(VFD_1_Current_Real,VFD_1_Tot.EI) ];
   // READ CURRENT FROM PF70ER - RIGHT DRYER VFD
   44: EQU(3,INTERRUPT_INDEX)[MSG(PF70ER_Message) ,DIV(VFD_2_Current,100,VFD_2_Current_Real) MOV(VFD_2_Current_Real,VFD_2_Tot.EI) ];
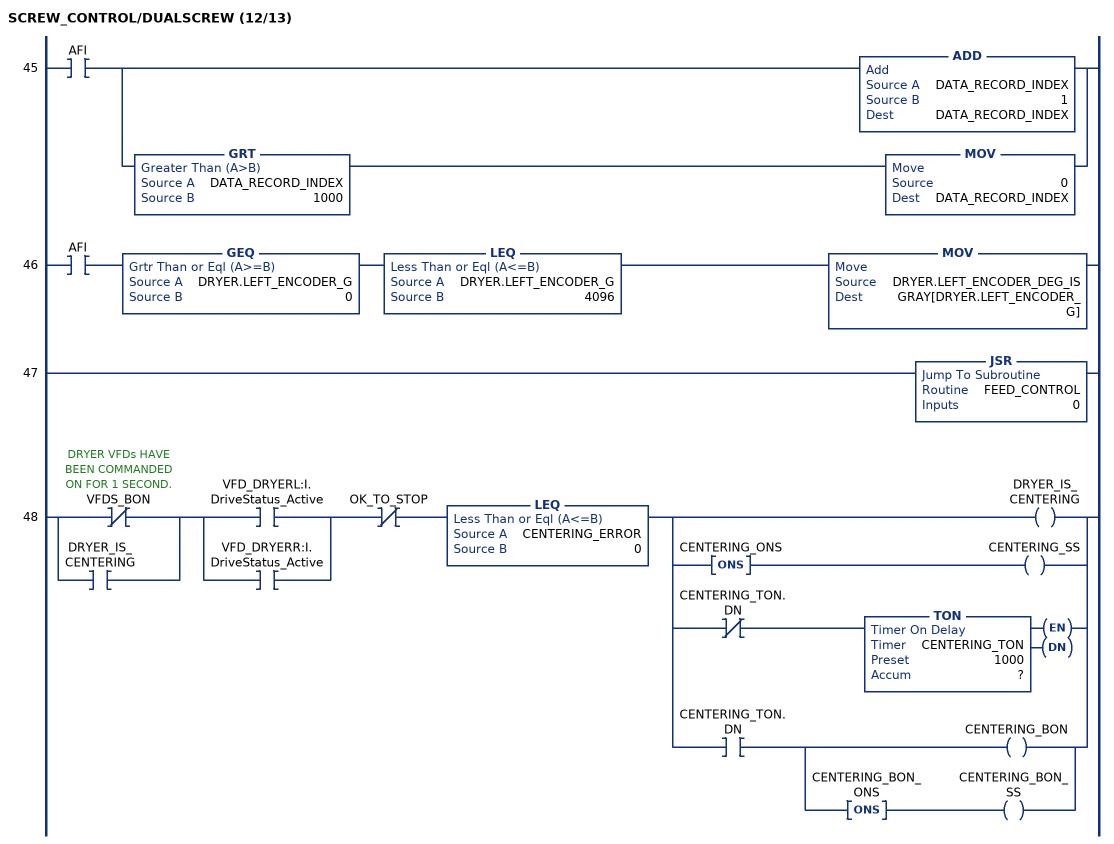
   45: XIC(AFI)[ADD(DATA_RECORD_INDEX,1,DATA_RECORD_INDEX) ,GRT(DATA_RECORD_INDEX,1000) MOV(0,DATA_RECORD_INDEX) ];
   46: XIC(AFI)GEQ(DRYER.LEFT_ENCODER_G,0)LEQ(DRYER.LEFT_ENCODER_G,4096)MOV(DRYER.LEFT_ENCODER_DEG_IS,GRAY[DRYER.LEFT_ENCODER_G]);
   47: JSR(FEED_CONTROL,0);
   48: [XIO(VFDS_BON) ,XIC(DRYER_IS_CENTERING) ][XIC(VFD_DRYERL:I.DriveStatus_Active) ,XIC(VFD_DRYERR:I.DriveStatus_Active) ]XIO(OK_TO_STOP)LEQ(CENTERING_ERROR,0)[OTE(DRYER_IS_CENTERING) ,ONS(CENTERING_ONS) OTE(CENTERING_SS) ,XIO(CENTERING_TON.DN) TON(CENTERING_TON,?,?) ,XIC(CENTERING_TON.DN) [OTE(CENTERING_BON) ,ONS(CENTERING_BON_ONS) OTE(CENTERING_BON_SS) ] ];
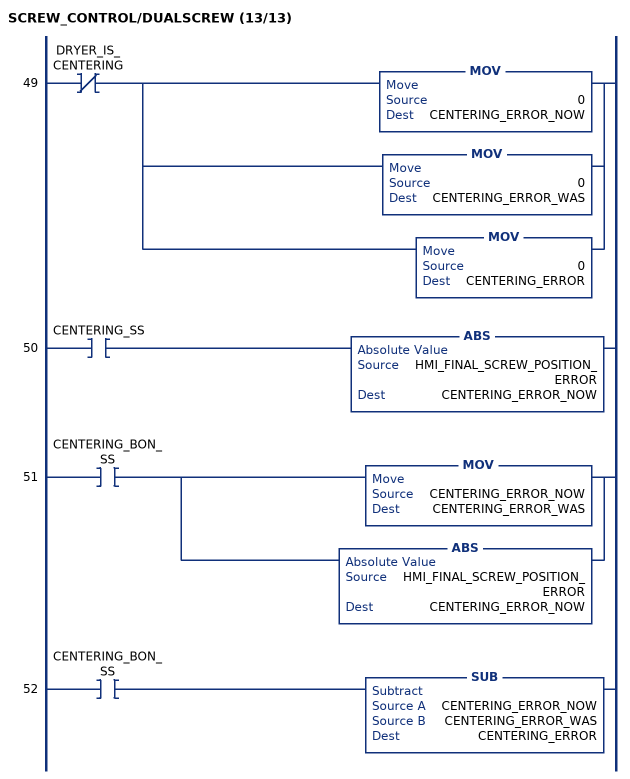
   49: XIO(DRYER_IS_CENTERING)[MOV(0,CENTERING_ERROR_NOW) ,MOV(0,CENTERING_ERROR_WAS) ,MOV(0,CENTERING_ERROR) ];
   50: XIC(CENTERING_SS)ABS(HMI_FINAL_SCREW_POSITION_ERROR,CENTERING_ERROR_NOW);
   51: XIC(CENTERING_BON_SS)[MOV(CENTERING_ERROR_NOW,CENTERING_ERROR_WAS) ,ABS(HMI_FINAL_SCREW_POSITION_ERROR,CENTERING_ERROR_NOW) ];
   52: XIC(CENTERING_BON_SS)SUB(CENTERING_ERROR_NOW,CENTERING_ERROR_WAS,CENTERING_ERROR);
END_ROUTINE
